FUNCTION_BLOCK FB_CartCtrlInit EXTENDS FB_CartCtrlBase
VAR_INPUT
END_VAR
VAR_OUTPUT
END_VAR
VAR
END_VAR

// override this function in each exact controller
METHOD PROTECTED calcCmdJntPos : BOOL
VAR_IN_OUT CONSTANT
	// slave cart joint data
	i_slaveCart :FB_SlaveCart;
END_VAR
IF m_timePeriod > 1.0 THEN
	m_isFinished := true;
END_IF
END_METHOD

// override this function in each exact controller
// NOTICE: set joint control mode here, and do some initialization if needed
METHOD PUBLIC init : BOOL
VAR_IN_OUT CONSTANT
	i_slaveCart	:FB_SlaveCart;
END_VAR
VAR_IN_OUT 
	r_cartCtrlCmd :ST_SlaveArmCtrlCmds;
END_VAR
SUPER^.init(i_slaveCart,r_cartCtrlCmd);

// update commands to arm
copyCmds(r_cartCtrlCmd);
END_METHOD

END_FUNCTION_BLOCK

(* stored: Version 1.1.0.1, ProductVersion 3.1.4024.11
   POU FB_CartCtrlInit: Id {4e4d6d84-764b-422d-abbc-80316d089754}, SpecialFunc None
   Method calcCmdJntPos: Id {e82173d7-fed9-4431-b4f7-e593032abfa8}
   Method init: Id {08fbbc2f-884e-4360-8758-0ef84c282cba} *)
